TYPE ST_WriteSingleOffsetData_Status EXTENDS ST_StatusBasic :
STRUCT
END_STRUCT
END_TYPE

(* stored: Version 1.1.0.1, ProductVersion 3.1.4024.13
   DUT ST_WriteSingleOffsetData_Status: Id {ba34a339-7912-4e86-8790-aa385ba3778c} *)
